Staubli VAL3: OnEvent18.pgx

program OnEvent18()
  local bool l_bBool
begin
  //-----------------------------------------------------------------------
  //Header begin
  //LasMAN3.7
  //Description of program
  //
  //Input parameters
  //
  //Output paramaters
  //Example
  //  call OnEvent1()
  //History
  //  Creation : 2013-06-23  y.ye@staubli.com
  //Header end
  //-----------------------------------------------------------------------
  resetMotion()
  //      call UI:Control_YesNO("确定替换空白的调试文件吗?",l_bBool)
  //      if l_bBool
  //        call TxtFile:SaveNewProduct(l_bBool)
  //
  //      endIf
  call Teach:TeachSyncAxis()
  DataBase:nInterfaceType=9
end
